(* PLC project marvel_unit, Institute of Astronomy Onto 0.0.1 *)
(* stored: creationDateTime 2025-01-01T00:00:00.0, modificationDateTime 2025-01-01T00:00:00.0 *)

TYPE UnitParts : STRUCT
  {attribute 'TcHmiSymbol.Show'}
  dome : Dome;  (* The dome *)
  {attribute 'TcHmiSymbol.Show'}
  guiding : Guiding;  (* The guiding *)
  {attribute 'TcHmiSymbol.Show'}
  fem : Fem;  (* The front end module *)
  {attribute 'TcHmiSymbol.Show'}
  telescope : Telescope;  (* The telescope *)
  {attribute 'TcHmiSymbol.Show'}
  configManager : ConfigManager;  (* The config manager (to load/save/activate configuration data) *)
END_STRUCT;
END_TYPE

TYPE UnitProcesses : STRUCT
  {attribute 'TcHmiSymbol.Show'}
  initialize : Process;  (* Start initializing the unit *)
  {attribute 'TcHmiSymbol.Show'}
  point : PointAlphaDeltaProcess;  (* Point the telescope and dome *)
  {attribute 'TcHmiSymbol.Show'}
  stop : Process;  (* Stop the rotation movement and/or tracking *)
END_STRUCT;
END_TYPE

TYPE UnitStatuses : STRUCT
  {attribute 'OPC.UA.DA' := '1'}
  {attribute 'OPC.UA.DA.Access' := '1'}
  {attribute 'TcHmiSymbol.Show'}
  init : InitializationStatus;
  {attribute 'OPC.UA.DA' := '1'}
  {attribute 'OPC.UA.DA.Access' := '1'}
  {attribute 'TcHmiSymbol.Show'}
  health : HealthStatus;
  {attribute 'OPC.UA.DA' := '1'}
  {attribute 'OPC.UA.DA.Access' := '1'}
  {attribute 'TcHmiSymbol.Show'}
  busy : BusyStatus;
END_STRUCT;
END_TYPE

TYPE UnitConfig : STRUCT
  {attribute 'TcHmiSymbol.Show'}
  dome : DomeConfig;  (* Dome config of a Marvel unit *)
  {attribute 'TcHmiSymbol.Show'}
  telescope : TelescopeConfig;  (* Telescope config of a Marvel unit *)
  {attribute 'TcHmiSymbol.Show'}
  guiding : GuidingConfig;  (* Guiding config of a Marvel unit *)
  {attribute 'TcHmiSymbol.Show'}
  fem : FemConfig;  (* Front End Module config of a Marvel unit *)
END_STRUCT;
END_TYPE

TYPE M_SM_Unit : STRUCT
  {attribute 'OPC.UA.DA' := '1'}
  {attribute 'OPC.UA.DA.Access' := '1'}
  {attribute 'TcHmiSymbol.Show'}
  number : USINT;
  {attribute 'OPC.UA.DA' := '1'}
  {attribute 'OPC.UA.DA.Access' := '3'}
  {attribute 'TcHmiSymbol.Show'}
  editableConfig : UnitConfig;
  {attribute 'OPC.UA.DA' := '1'}
  {attribute 'OPC.UA.DA.Access' := '1'}
  {attribute 'TcHmiSymbol.Show'}
  actualStatus : STRING;
  {attribute 'OPC.UA.DA' := '1'}
  {attribute 'OPC.UA.DA.Access' := '1'}
  {attribute 'TcHmiSymbol.Show'}
  config : UnitConfig;
  {attribute 'OPC.UA.DA' := '1'}
  {attribute 'OPC.UA.DA.Access' := '1'}
  {attribute 'TcHmiSymbol.Show'}
  targetAlpha : AngularPosition;
  {attribute 'OPC.UA.DA' := '1'}
  {attribute 'OPC.UA.DA.Access' := '1'}
  {attribute 'TcHmiSymbol.Show'}
  targetDelta : AngularPosition;
  {attribute 'OPC.UA.DA' := '1'}
  {attribute 'TcHmiSymbol.Show'}
  stat : UnitStatuses;
  {attribute 'OPC.UA.DA' := '1'}
  {attribute 'TcHmiSymbol.Show'}
  parts : M_SM_UnitParts;
  {attribute 'OPC.UA.DA' := '1'}
  {attribute 'TcHmiSymbol.Show'}
  proc : M_SM_UnitProcesses;
END_STRUCT;
END_TYPE

TYPE M_SM_UnitParts : STRUCT
  {attribute 'TcHmiSymbol.Show'}
  dome : M_Dome;
  {attribute 'TcHmiSymbol.Show'}
  guiding : M_Guiding;
  {attribute 'TcHmiSymbol.Show'}
  fem : M_Fem;
  {attribute 'TcHmiSymbol.Show'}
  telescope : M_Telescope;
  {attribute 'TcHmiSymbol.Show'}
  configManager : M_ConfigManager;
END_STRUCT;
END_TYPE

TYPE M_SM_UnitProcesses : STRUCT
  {attribute 'TcHmiSymbol.Show'}
  initialize : M_Process;
  {attribute 'TcHmiSymbol.Show'}
  point : M_PointAlphaDeltaProcess;
  {attribute 'TcHmiSymbol.Show'}
  stop : M_Process;
END_STRUCT;
END_TYPE

FUNCTION_BLOCK SM_Unit
  VAR_INPUT
    {attribute 'OPC.UA.DA' := '1'}
    {attribute 'OPC.UA.DA.Access' := '1'}
    number : USINT;  (* Number of the unit (1-4) *)
    {attribute 'OPC.UA.DA' := '1'}
    {attribute 'OPC.UA.DA.Access' := '3'}
    editableConfig : UnitConfig;  (* Editable configuration of the unit *)
  END_VAR
  VAR_OUTPUT
    {attribute 'OPC.UA.DA' := '1'}
    {attribute 'OPC.UA.DA.Access' := '1'}
    actualStatus : STRING(50);  (* Current status description *)
    {attribute 'OPC.UA.DA' := '1'}
    {attribute 'OPC.UA.DA.Access' := '1'}
    config : UnitConfig;  (* Active configuration of the unit *)
    {attribute 'OPC.UA.DA' := '1'}
    {attribute 'OPC.UA.DA.Access' := '1'}
    targetAlpha : AngularPosition;  (* The target alpha coordinate (Right Ascention) *)
    {attribute 'OPC.UA.DA' := '1'}
    {attribute 'OPC.UA.DA.Access' := '1'}
    targetDelta : AngularPosition;  (* The target delta coordinate (Declination) *)
    {attribute 'OPC.UA.DA' := '1'}
    stat : UnitStatuses;  (* Statuses of the state machine *)
    {attribute 'OPC.UA.DA' := '1'}
    parts : UnitParts;  (* Parts of the state machine *)
    {attribute 'OPC.UA.DA' := '1'}
    proc : UnitProcesses;  (* Processes of the state machine *)
  END_VAR
  VAR_IN_OUT
    {attribute 'OPC.UA.DA' := '0'}
    operator_ref : OperatorStatus;  (* Reference to the operator (observer/tech) *)
    {attribute 'OPC.UA.DA' := '0'}
    activity_ref : ActivityStatus;  (* Shared activity status *)
    {attribute 'OPC.UA.DA' := '0'}
    services_ref : Services;  (* Shared services *)
  END_VAR

            parts.dome(
    operator_ref := operator_ref,
    activity_ref := activity_ref,
    services_ref := services_ref,
    config_ref := config.dome,
    telescopeAzi_ref := parts.telescope.actAzi);
parts.guiding(
    number := number,
    operator_ref := operator_ref,
    activity_ref := activity_ref,
    services_ref := services_ref,
    camera_ref := parts.fem.parts.guideCam,
    config_ref := config.guiding);
parts.fem(
    number := number,
    operator_ref := operator_ref,
    activity_ref := activity_ref,
    services_ref := services_ref,
    config_ref := config.fem);
parts.telescope(
    operator_ref := operator_ref,
    activity_ref := activity_ref,
    services_ref := services_ref,
    config_ref := config.telescope);
parts.configManager( isEnabled := operator_ref = OperatorStatus.tech );
stat.health := F_HealthStatus(
    superState := NOT(stat.init = InitializationStatus.shutdown),
    isGood := (NOT(stat.init = InitializationStatus.initializingFailed)) AND (((parts.dome.stat.health = HealthStatus.good) OR (parts.dome.stat.health = HealthStatus.warning)) AND (((parts.telescope.stat.health = HealthStatus.good) OR (parts.telescope.stat.health = HealthStatus.warning)) AND (((parts.fem.stat.health = HealthStatus.good) OR (parts.fem.stat.health = HealthStatus.warning)) AND ((parts.configManager.stat.health = HealthStatus.good) OR (parts.configManager.stat.health = HealthStatus.warning))))),
    hasWarning := (parts.dome.stat.health = HealthStatus.warning) OR ((parts.telescope.stat.health = HealthStatus.warning) OR ((parts.fem.stat.health = HealthStatus.warning) OR (parts.configManager.stat.health = HealthStatus.warning))));
stat.busy := F_BusyStatus(
    superState := NOT(stat.init = InitializationStatus.shutdown),
    isBusy := (parts.dome.stat.busy = BusyStatus.busy) OR ((parts.telescope.stat.busy = BusyStatus.busy) OR ((parts.fem.stat.busy = BusyStatus.busy) OR (parts.configManager.stat.busy = BusyStatus.busy))));
proc.initialize( isEnabled := NOT(stat.init = InitializationStatus.initializing) );
proc.point( isEnabled := (stat.init = InitializationStatus.initialized) AND (proc.point.stat.busy = BusyStatus.idle) );
proc.stop( isEnabled := parts.telescope.proc.abortSlew.isEnabled OR parts.dome.proc.stop.isEnabled );

          

METHOD _copyFromModel_SM_Unit
  VAR_IN_OUT
    {attribute 'OPC.UA.DA' := '0'}
    model : M_SM_Unit;
  END_VAR
                  THIS^.editableConfig := model.editableConfig;
THIS^.parts.dome._copyFromModel_Dome( model := model.parts.dome );
THIS^.parts.guiding._copyFromModel_Guiding( model := model.parts.guiding );
THIS^.parts.fem._copyFromModel_Fem( model := model.parts.fem );
THIS^.parts.telescope._copyFromModel_Telescope( model := model.parts.telescope );
THIS^.parts.configManager._copyFromModel_ConfigManager( model := model.parts.configManager );
THIS^.proc.initialize._copyFromModel_Process( model := model.proc.initialize );
THIS^.proc.point._copyFromModel_PointAlphaDeltaProcess( model := model.proc.point );
THIS^.proc.stop._copyFromModel_Process( model := model.proc.stop );

                
END_METHOD

METHOD _copyToModel_SM_Unit
  VAR_IN_OUT
    {attribute 'OPC.UA.DA' := '0'}
    model : M_SM_Unit;
  END_VAR
                  model.number := THIS^.number;
model.editableConfig := THIS^.editableConfig;
model.actualStatus := THIS^.actualStatus;
model.config := THIS^.config;
model.targetAlpha := THIS^.targetAlpha;
model.targetDelta := THIS^.targetDelta;
model.stat := THIS^.stat;
THIS^.parts.dome._copyToModel_Dome( model := model.parts.dome );
THIS^.parts.guiding._copyToModel_Guiding( model := model.parts.guiding );
THIS^.parts.fem._copyToModel_Fem( model := model.parts.fem );
THIS^.parts.telescope._copyToModel_Telescope( model := model.parts.telescope );
THIS^.parts.configManager._copyToModel_ConfigManager( model := model.parts.configManager );
THIS^.proc.initialize._copyToModel_Process( model := model.proc.initialize );
THIS^.proc.point._copyToModel_PointAlphaDeltaProcess( model := model.proc.point );
THIS^.proc.stop._copyToModel_Process( model := model.proc.stop );

                
END_METHOD
END_FUNCTION_BLOCK
